// TIA Portal V15.1 export
// export: Created 2020-06-12T07:35:51.4912109Z, ExportSetting None, DisplayName Totally Integrated Automation Portal, DisplayVersion V15.1, DisplayName TIA Portal Openness, DisplayVersion V15.1, DisplayName STEP 7 Professional, DisplayVersion V15.1, DisplayName STEP 7 Safety, DisplayVersion V15.1, DisplayName WinCC Advanced, DisplayVersion V15.1
FUNCTION "MELT_CPF_VP" : Void   // FC170, FBD
TITLE = Speed(Resistance) controller treat
{ S7_Optimized_Access := 'TRUE' }
// stored: SetENOAutomatically False
   VAR_TEMP
      tBool : Bool;
      tSetIndex2 : Int;
      tSelect : Bool;
      tUseCh2 : Bool;
      tPV : Real;
      tSP : Real;
      tUmin : Real;
      tUdir : Real;
      tUset1 : Real;
      tUset0 : Real;
      tIsOn0 : Bool;
      tIsOn1 : Bool;
      tIset : Real;
      tUdrop : Real;
      tUset2 : Real;
      tUmax : Real;
   END_VAR
BEGIN

REGION Network 1: Select the parameter set
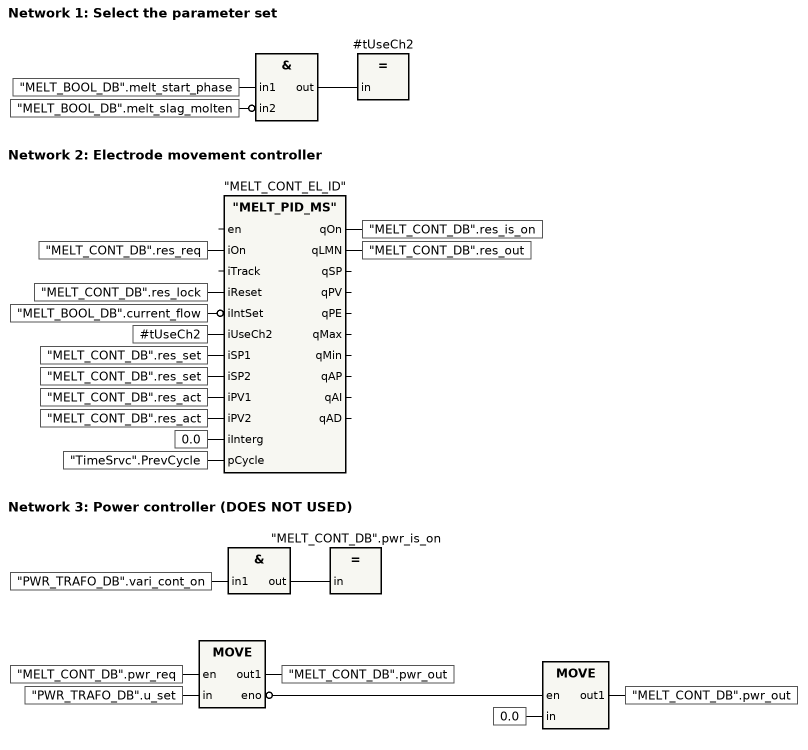
   #tUseCh2 := "MELT_BOOL_DB".melt_start_phase AND NOT "MELT_BOOL_DB".melt_slag_molten;
END_REGION

REGION Network 2: Electrode movement controller
   "MELT_CONT_EL_ID"(iOn := "MELT_CONT_DB".res_req,   // "MELT_PID_MS"
                     iReset := "MELT_CONT_DB".res_lock,
                     iIntSet := NOT "MELT_BOOL_DB".current_flow,
                     iUseCh2 := #tUseCh2,
                     iSP1 := "MELT_CONT_DB".res_set,
                     iSP2 := "MELT_CONT_DB".res_set,
                     iPV1 := "MELT_CONT_DB".res_act,
                     iPV2 := "MELT_CONT_DB".res_act,
                     iInterg := 0.0,
                     pCycle := "TimeSrvc".PrevCycle,
                     qOn => "MELT_CONT_DB".res_is_on,
                     qLMN => "MELT_CONT_DB".res_out);
END_REGION

REGION Network 3: Power controller (DOES NOT USED)
   // The power controller is implemented as part of transformer controller.
   // Well, we do some trick to keep the variables state consistent
   "MELT_CONT_DB".pwr_is_on := "PWR_TRAFO_DB".vari_cont_on;
   IF "MELT_CONT_DB".pwr_req THEN "MELT_CONT_DB".pwr_out := "PWR_TRAFO_DB".u_set; END_IF;
   IF NOT "MELT_CONT_DB".pwr_req THEN "MELT_CONT_DB".pwr_out := 0.0; END_IF;
END_REGION
END_FUNCTION
